TYPE E_AlarmState :
(
    ALARM_INACTIVE      := 0,
    ALARM_ACTIVE        := 1,
    ALARM_ACKNOWLEDGED  := 2,
    ALARM_CLEARED       := 3
);
END_TYPE

(* stored: Version 1.1.0.1
   DUT E_AlarmState: Id {7BC7FEB8-00CC-F308-D5EB-A13099180ED6} *)
